{attribute 'qualified_only'}
{attribute 'strict'}
{attribute 'to_string'}
TYPE ELopendeBandStatus :
(
	Stopped := 0,
	Starting,
	Stopping,
	Running,
	Error
);
END_TYPE

(* stored: Version 1.1.0.1
   DUT ELopendeBandStatus: Id {75141f50-25e9-4d67-8389-7fe1d1bef885} *)
